// TIA Portal V19 export
DATA_BLOCK "Loop1"   // DB192
{ DB_Accessible_From_OPC_UA := 'FALSE' }
// stored: DBAccessibleFromOPCUA false, InstanceOfName SmartLoopControl, InstanceOfType FB
"SmartLoopControl"
   // VAR_INPUT
   //    AreaInterfaceEntry : "AreaInterface";
   //    AreaInterfaceExit : "AreaInterface";
   //    DataIn : Struct
   //       Pb_StartStop : Bool;
   //       Pb_Start : Bool;
   //       Pb_Stop : Bool;
   //       SensorEntryMaterialPresence : Bool;
   //       SensorExitMaterialPresence : Bool;
   //       SensorExitEnableUseEncoder : Bool;
   //       SensorNotLoopMinHigh : Bool;
   //       SensorLoopMaxLow_Or_TPEntry : Bool;
   //       SensorLoopMaxLow_Or_TPExit : Bool;
   //       PlugConnected : Bool;
   //    END_STRUCT;
   //    CIn : "SmartLoopControl_CIn";
   //    Config : Struct
   //       PitTables_Exist : Bool;
   //       Entry_PercentagePosError : LReal;
   //       Exit_PercentagePosError : LReal;
   //       Delay_CheckNoEntryBkwEnable : Time;
   //       Delay_CheckNoEntryFwdEnable : Time;
   //       Delay_CheckNoExitBkwEnable : Time;
   //       Delay_CheckNoExitFwdEnable : Time;
   //    END_STRUCT;
   // END_VAR
   // VAR_OUTPUT
   //    MachineInterfaceEntry : "MachineInterface";
   //    MachineInterfaceExit : "MachineInterface";
   //    COut : "SmartLoopControl_COut";
   //    DataOut : Struct
   //       LampSystemOn : Bool;
   //    END_STRUCT;
   // END_VAR
   // VAR_IN_OUT
   //    PersistentValues : Struct
   //       Par : "SmartLoopControl_Par";
   //    END_STRUCT;
   // END_VAR
   // VAR
   //    Ctrl : Struct
   //       RstAlarms : Bool;
   //       StopInPhase : Bool;
   //       StopProgrammed : Bool;
   //       StopAborting : Bool;
   //       ForceSyncFirstStart : Bool;
   //       ForceSyncMinHigh : Bool;
   //       ForceSyncCyclic : Bool;
   //       ForceSyncExt : Bool;
   //       ForceSync : Bool;
   //       Sync_Exe : Bool;
   //       Sync_EntryReduceOrStopFeed : Bool;
   //       Sync_ExitReduceOrStopFeed : Bool;
   //       MeasuringEnable : Bool;
   //       Entry_EnableFeedBkw : Bool;
   //       Entry_EnableFeedFwd : Bool;
   //       Exit_EnableFeedBkw : Bool;
   //       Exit_EnableFeedFwd : Bool;
   //       Entry_VelocityOverride : LReal;
   //       Exit_VelocityOverride : LReal;
   //       Exit_MaxAllowableFeedFwd : LReal;
   //    END_STRUCT;
   //    Sts : Struct
   //       IsStandstill : Bool;
   //       AlarmsPresence : Bool;
   //       WarningsPresence : Bool;
   //       SensorsMaxLow_OFF : Bool;
   //       SensorsMaxLow_ON : Bool;
   //       LoopMaterialCounterValid : Bool;
   //       SynchroRunning : Bool;
   //       CheckSensorCatchIsOn : Bool;
   //       CheckSensorLooseIsOn : Bool;
   //       WorkModeMatCounter : Bool;
   //       WorkModeSensors : Bool;
   //       SystemOn : Bool;
   //       MinHighReached : Bool;
   //       SynchroDone : Bool;
   //       CntFeedIncValid : Bool;
   //       AntiRepetitionForceSyncExt : Bool;
   //       Entry_MeasuringValuePosAxValid : Bool;
   //       Exit_MeasuringValuePosAxValid : Bool;
   //       Entry_MeasuringValueMatCounterValid : Bool;
   //       Exit_MeasuringValueMatCounterValid : Bool;
   //       SynchroDoneTof2s : Bool;
   //       MaxLowReached : Bool;
   //       SelectedPosStopMaxLow : LReal;
   //       SelectedOverrideScaling : LReal;
   //       LoopMaterialCounter : LReal;
   //       DifferenceInc : LReal;
   //       CntFeedIncPrevious : LReal;
   //       MissingToCyclicSync : LReal;
   //       SyncroMemLoopMaterialCounter : LReal;
   //       AntiRepetitionForceSyncExtSaveEntryMatCounter : LReal;
   //       AntiRepetitionForceSyncExtSaveExitMatCounter : LReal;
   //       EncEntry_MeasuringValuePosAx : LReal;
   //       EncExit_MeasuringValuePosAx : LReal;
   //       EncEntry_MeasuringValueMatCounter : LReal;
   //       EncExit_MeasuringValueMatCounter : LReal;
   //       LoopMaterialCounterOffset : LReal;
   //       LoopMaterialMissingToMaxLow : LReal;
   //       LoopMaterialMissingToMinHigh : LReal;
   //       Cases_Entry_VelocityOverride : UInt;
   //       Cases_Exit_VelocityOverride : UInt;
   //       Cases_Exit_MaxFeed : UInt;
   //       WorkMode : UInt;
   //    END_STRUCT;
   //    Wng : Struct
   //       NoAutReady : Bool;
   //       MeasInputsXORMeasuringValue : Bool;
   //       TimeOutCalculateLoopCounterOffset : Bool;
   //       SensorEnableEncIsOff : Bool;
   //       Entry_MatCounterNotValid : Bool;
   //       Exit_MatCounterNotValid : Bool;
   //       NotSystemOn : Bool;
   //       MinHighReached : Bool;
   //       SyncNeedToLooseSensor : Bool;
   //       SyncNeedToCatchSensor : Bool;
   //       Entry_NoBkwEnable : Bool;
   //       Entry_NoFwdEnable : Bool;
   //       Exit_NoBkwEnable : Bool;
   //       Exit_NoFwdEnable : Bool;
   //    END_STRUCT;
   //    Alr : Struct
   //       MeasInputsXORInputState : Bool;
   //       Entry_MatCounterLooseOfValidState : Bool;
   //       Exit_MatCounterLooseOfValidState : Bool;
   //       SensorError : Bool;
   //       PlugNotConnected : Bool;
   //       SyncSensorNotCatch : Bool;
   //       SyncSensorNotLoose : Bool;
   //       Entry_NoCounterMove : Bool;
   //       Exit_NoCounterMove : Bool;
   //    END_STRUCT;
   //    tonCheckMeasInputStateXOR : TON_TIME;
   //    tonDelaySensorMaxLowLoose { S7_SetPoint := 'True'} : TON_TIME;
   //    tonDelaySensorMaxLowCatch { S7_SetPoint := 'True'} : TON_TIME;
   //    tonCheckNoEntryCounterMove { S7_SetPoint := 'True'} : TON_TIME;
   //    tonCheckNoExitCounterMove { S7_SetPoint := 'True'} : TON_TIME;
   //    tonEnableForceSyncCyclic { S7_SetPoint := 'True'} : TON_TIME;
   //    tonSynchIdle { S7_SetPoint := 'True'} : TON_TIME;
   //    tonCheckBothMeasuringDone { S7_SetPoint := 'True'} : TON_TIME;
   //    tonTimeOutCalculateCounterOffset { S7_SetPoint := 'True'} : TON_TIME;
   //    tonSynchAutoReset { S7_SetPoint := 'True'} : TON_TIME;
   //    tof2sSynchroDone { S7_SetPoint := 'True'} : TON_TIME;
   //    tonRstMaterialCounterValid { S7_SetPoint := 'True'} : TON_TIME;
   //    tonSetMaxLow { S7_SetPoint := 'True'} : TON_TIME;
   //    tonRstMaxLow { S7_SetPoint := 'True'} : TON_TIME;
   //    tonCheckNoEntryBkwEnable { S7_SetPoint := 'True'} : TON_TIME;
   //    tonCheckNoEntryFwdEnable { S7_SetPoint := 'True'} : TON_TIME;
   //    tonCheckNoExitBkwEnable { S7_SetPoint := 'True'} : TON_TIME;
   //    tonCheckNoExitFwdEnable { S7_SetPoint := 'True'} : TON_TIME;
   //    SynchCycle { S7_SetPoint := 'True'} : UInt;
   //    CheckSensorCatchSaveLoopMaterialCounter : LReal;
   //    CheckSensorCatchFeeding : LReal;
   //    CheckSensorLooseSaveLoopMaterialCounter : LReal;
   //    CheckSensorLooseFeeding : LReal;
   //    AuxPbStartStopOneShot { S7_SetPoint := 'True'} : Bool;
   //    AuxSyncFirstStartOneShot : Bool;
   //    ModeMatCounterAndSystemOn : Bool;
   //    MinHighCumulative : Bool;
   //    AuxSyncMinHighOneShot : Bool;
   //    Entry_SaveMesInpID : UInt;
   //    Exit_SaveMesInpID : UInt;
   //    Check_Entry_Velocity { S7_SetPoint := 'True'} : "Check_Axis_Velocity";
   //    Check_Exit_Velocity { S7_SetPoint := 'True'} : "Check_Axis_Velocity";
   // END_VAR
BEGIN
END_DATA_BLOCK
